RoboDK station: RBT23CB016_Palletizing_2Finger_Gripper - Copy.rdk

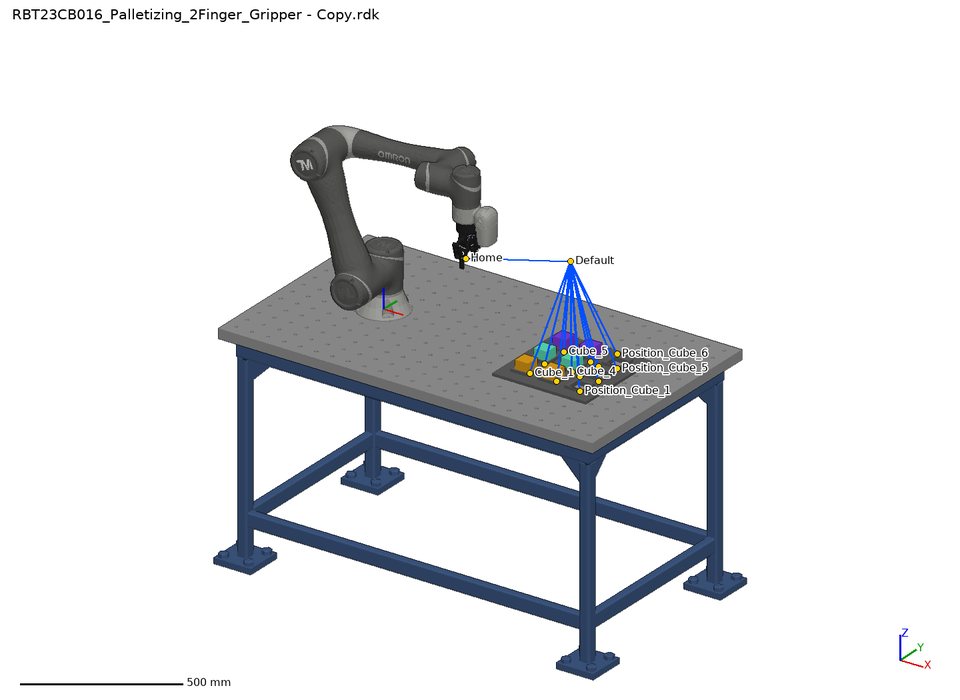
[picture v0: the station drawn from its stored meshes, robots at their saved joint values, targets as dots, program paths as lines]
Station RBT23CB016_Palletizing_2Finger_Gripper (saved by RoboDK 5.9.2). Poses are relative to the parent item; angles as X-Y-Z fixed-axis rotations.
  - frame Base at (0, 1000, 0) mm
    - robot Omron TM5-900: 6 axes, payload 4 kg, reach 900 mm, repeatability 0.05 mm, weight 22.6 kg
        modified DH rows (alpha deg, a mm, theta deg, d mm): 0, 0, 0, 145.2; 90, 0, 90, 0; 0, 429, 0, 0; 0, 411, -90, 122.3; -90, 0, 0, 106.5; 90, 0, 180, 114.15
        joint limits [-270, -180, -155, -180, -180, -270] to [270, 180, 155, 180, 180, 270]; home [0, 0, 90, -90, 90, 0]; saved at [3.322, -19.705, 107.836, 2.129, 90.143, 3.315]
      - tool RobotiQ 2F-85 Gripper (Closed), TCP at (0, 0, 130) mm, size 134.4 x 75 x 157.6 mm
    - target Home (Cartesian target) at (377.95, -99.96, 317.85) mm, rotated rx -179.73 ry -0.13 rz 90.01 deg; joints [3.322, -19.705, 107.836, 2.129, 90.143, 3.315] of Omron TM5-900
    - target Default (Cartesian target) at (704.21, -9.35, 363.79) mm, rotated rx -179.75 ry -0.15 rz 95.85 deg; joints [9.18, 25.441, 53.933, 10.871, 90.168, 3.334] of Omron TM5-900
    - target Cube_1 (Cartesian target) at (616.33, -99.22, -6.12) mm, rotated rx -179.73 ry -0.13 rz 90.01 deg; joints [2.098, 28.982, 104.334, -43.054, 90.137, 2.091] of Omron TM5-900
    - target Cube_2 (Cartesian target) at (716.33, -99.22, -6.12) mm, rotated rx -179.73 ry -0.13 rz 90.01 deg; joints [1.804, 39.424, 85.972, -35.133, 90.135, 1.798] of Omron TM5-900
    - target Cube_3 (Cartesian target) at (616.32, -19.22, -6.12) mm, rotated rx -179.73 ry -0.13 rz 90.01 deg; joints [9.585, 28.2, 105.663, -43.62, 90.17, 9.579] of Omron TM5-900
    - target Cube_4 (Cartesian target) at (716.33, -19.22, -6.12) mm, rotated rx -179.73 ry -0.13 rz 90.01 deg; joints [8.233, 38.696, 87.296, -35.745, 90.164, 8.227] of Omron TM5-900
    - target Cube_5 (Cartesian target) at (615.46, 82.22, -6.99) mm, rotated rx -179.73 ry -0.13 rz 90.01 deg; joints [18.885, 28.718, 104.968, -43.473, 90.207, 18.878] of Omron TM5-900
    - target Cube_6 (Cartesian target) at (715.33, 82.24, -12.73) mm, rotated rx -179.73 ry -0.13 rz 90.01 deg; joints [16.27, 39.591, 86.821, -36.191, 90.197, 16.263] of Omron TM5-900
    - target Position_Cube_1 (Cartesian target) at (813.96, -115.89, -4.98) mm, rotated rx -179.73 ry -0.13 rz 90.01 deg; joints [0.413, 51.364, 63.589, -24.686, 90.129, 0.407] of Omron TM5-900
    - target Position_Cube_2 (Cartesian target) at (813.96, -115.88, 45.02) mm, rotated rx -179.73 ry -0.13 rz 90.01 deg; joints [0.413, 48.492, 61.401, -19.626, 90.129, 0.407] of Omron TM5-900
    - target Position_Cube_3 (Cartesian target) at (814.56, -16.66, -11.8) mm, rotated rx -179.73 ry -0.13 rz 90.01 deg; joints [7.413, 50.796, 65.731, -26.278, 90.16, 7.407] of Omron TM5-900
    - target Position_Cube_4 (Cartesian target) at (814.56, -16.66, 38.2) mm, rotated rx -179.73 ry -0.13 rz 90.01 deg; joints [7.413, 47.79, 63.708, -21.248, 90.16, 7.407] of Omron TM5-900
    - target Position_Cube_5 (Cartesian target) at (815.46, 82.22, -6.99) mm, rotated rx -179.73 ry -0.13 rz 90.01 deg; joints [14.282, 51.129, 64.356, -25.257, 90.189, 14.275] of Omron TM5-900
    - target Position_Cube_6 (Cartesian target) at (815.46, 82.22, 43.01) mm, rotated rx -179.73 ry -0.13 rz 90.01 deg; joints [14.282, 48.213, 62.221, -20.205, 90.189, 14.275] of Omron TM5-900
    - target Target 15 (Cartesian target) at (377.95, -99.96, 317.85) mm, rotated rx -179.73 ry -0.13 rz 90.01 deg; joints [3.322, -19.705, 107.836, 2.129, 90.142, 3.315] of Omron TM5-900
    - object Table 1400x800x800mm at (0, 0, 0) mm, size 1420 x 820 x 800 mm, geometry from Table-1400x800x800mm.sld
    - object Pallete at (539.16, -191.28, 0) mm, size 350 x 350 x 20 mm, geometry from Pallete  (1).step
    - object C4 at (537.95, -87.21, 43.57) mm, rotated rx 179.87 ry 0.27 rz 90.01 deg, size 50 x 50 x 50 mm, geometry from Cube-50mm.sld
    - object C3 at (539.16, -191.28, 0) mm, size 50 x 50 x 50 mm, geometry from Cube-50mm.sld
    - object C2 at (539.16, -191.28, 0) mm, size 50 x 50 x 50 mm, geometry from Cube-50mm.sld
    - object C1 at (539.16, -191.28, 0) mm, size 50 x 50 x 50 mm, geometry from Cube-50mm.sld
    - object C6 at (439.16, -91.28, 0) mm, size 50 x 50 x 50 mm, geometry from Cube-50mm.sld
    - object C5 at (439.16, -91.28, 0) mm, size 50 x 50 x 50 mm, geometry from Cube-50mm.sld
  - program Test_1 (41 instructions, listed below)
  - program Reset (1 instructions, listed below)
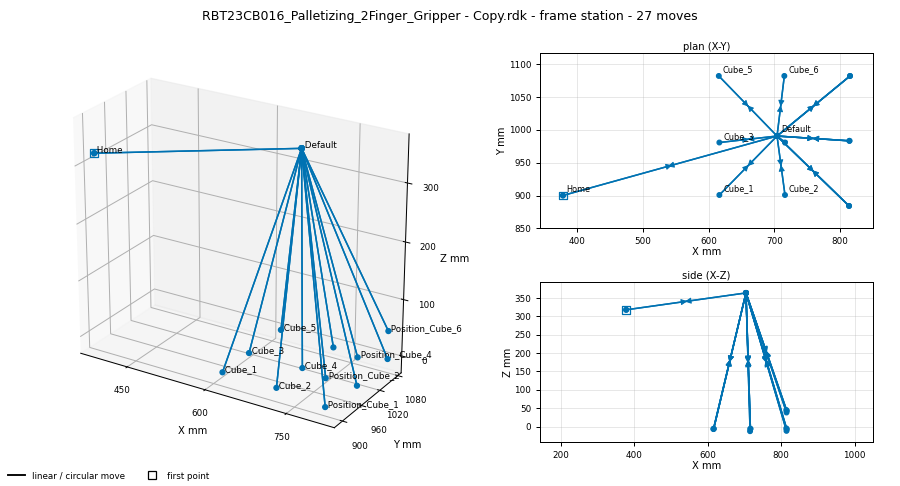
[picture p0: tool path of RBT23CB016_Palletizing_2Finger_Gripper - Copy.rdk in frame station, 27 of 27 moves have a stored position in this frame; points joined in program order, loops and branches not executed]

--- program Test_1 (robot Omron TM5-900) ---
  Set Ref.: Base
  MoveL (Home)
  MoveL (Default)
  MoveL (Cube_1)
  Attach to RobotiQ 2F-85 Gripper (Closed)
  MoveL (Default)
  MoveL (Position_Cube_1)
  Detach from RobotiQ 2F-85 Gripper (Closed)
  MoveL (Default)
  MoveL (Cube_2)
  Attach to RobotiQ 2F-85 Gripper (Closed)
  MoveL (Default)
  MoveL (Position_Cube_2)
  Detach from RobotiQ 2F-85 Gripper (Closed)
  MoveL (Default)
  MoveL (Cube_3)
  Attach to RobotiQ 2F-85 Gripper (Closed)
  MoveL (Default)
  MoveL (Position_Cube_3)
  Detach from RobotiQ 2F-85 Gripper (Closed)
  MoveL (Default)
  MoveL (Cube_4)
  Attach to RobotiQ 2F-85 Gripper (Closed)
  MoveL (Default)
  MoveL (Position_Cube_4)
  Detach from RobotiQ 2F-85 Gripper (Closed)
  MoveL (Default)
  MoveL (Cube_5)
  Attach to RobotiQ 2F-85 Gripper (Closed)
  MoveL (Default)
  MoveL (Position_Cube_5)
  Detach from RobotiQ 2F-85 Gripper (Closed)
  MoveL (Default)
  MoveL (Cube_6)
  Attach to RobotiQ 2F-85 Gripper (Closed)
  MoveL (Default)
  MoveL (Position_Cube_6)
  Detach from RobotiQ 2F-85 Gripper (Closed)
  MoveL (Default)
  MoveL (Home)
  Not defined

--- program Reset (robot Omron TM5-900) ---
  Replace objects
